// TIA Portal V15 export
// export: Created 2018-05-31T16:39:41.8318856Z, ExportSetting WithDefaults, WithReadOnly, DisplayName Totally Integrated Automation Portal, DisplayVersion V15, DisplayName TIA Portal Openness, DisplayVersion V15, DisplayName STEP 7 Professional, DisplayVersion V15, DisplayName WinCC Professional, DisplayVersion V15
DATA_BLOCK "LIC006_sp"   // DB1
{ S7_Optimized_Access := 'FALSE' }
VERSION : 0.1
// stored: AutoNumber true, CodeModifiedDate 2018-05-31T16:37:51.7325883Z, CompileDate 2018-05-31T16:37:51.7405888Z, CreationDate 2018-05-31T16:36:47.0278874Z, InterfaceModifiedDate 2018-05-31T16:37:42.3500517Z, IsConsistent true, IsKnowHowProtected false, IsOnlyStoredInLoadMemory false, IsPLCDB false, IsWriteProtectedInAS false, ModifiedDate 2018-05-31T16:37:51.7325883Z, ParameterModified 2018-05-31T16:37:42.3500517Z, StructureModified 2018-05-31T16:37:42.3500517Z
   VAR RETAIN
      Operator_Setpoint : Real;
      Set_SP : Bool;
      Output_Value : Real;
      Set_Output : Bool;
   END_VAR
BEGIN
END_DATA_BLOCK
